Staubli VAL3: tool.pjx

--- tool.pjx ---
Parameters version=s7.2.1 stackSize=5000 millimeterUnit=true
Program file=buildList.pgx
Program file=editAction.pgx
Program file=editTool.pgx
Program file=insertInstr.pgx
Program file=listAdd.pgx
Program file=loadPage.pgx
Program file=main.pgx
Program file=onBackSpace.pgx
Program file=onEnterEvent.pgx
Program file=onExit.pgx
Program file=onF1Event.pgx
Program file=onF2Event.pgx
Program file=onF3Event.pgx
Program file=onF4Event.pgx
Program file=onF5Event.pgx
Program file=onF6Event.pgx
Program file=onF7Event.pgx
Program file=onF8Event.pgx
Program file=onStart.pgx
Program file=refresh.pgx
Program file=refreshAction.pgx
Program file=refreshDynamic.pgx
Program file=refreshStatic.pgx
Data file=tool.dtx
Library alias=io path=Disk://io/io.pjx
Library alias=page path=Disk://kernel/template/page/page.pjx
Library alias=use path=Disk://kernel/userPage/userPage.pjx
Library alias=language path=Disk://kernel/language/language.pjx
Library alias=tcp path=Disk://kernel/tool/tool.pjx

--- tool.dtx ---
num nIndex
num nIndexTool
num nKey
public num nPage
num nRefresh
num nTime = 1
num nView
string sEvent
public string sItems
string sList
string sMenu
string sMessage
string sMenu8[8]
string sActionON[3]
string sActionOFF[3]
bool bButton[8]
bool bLarge

--- main.pgx ---
public program main()
  local tool l_tTool
  local num l_nSize
  local bool l_bSave
  local num l_nStatus
  local bool l_bToReset
  local bool l_bCalcolate
  local frame l_fNewWorld
begin
  // INIT
  call onStart()
  // LOOP UNTIL nKey=255
  do
    call tcp:getSize(l_nSize)
    call tcp:getTool(l_tTool,nIndexTool)
    call refresh()
    if l_bCalcolate
      $jogContext(l_tTool,world,0)
      l_bCalcolate=false
    endIf
    nKey=getKey()
    // tool setting

    // list....
    call use:listevent(nKey,nIndex,sEvent)
    nView=use:nView
    switch nKey
      case 263
        // BACKSPACE
        call onBackSpace(l_tTool)
        l_bCalcolate=true
        l_bSave=true
      break
      case 264
        // LEFT CLICK -1
        if nIndexTool>0
          nIndexTool=nIndexTool-1
          l_bSave=true
          l_bCalcolate=true
        endIf
      break
      case 268
        // RIGHT CLICK +1
        if nIndexTool<l_nSize-1
          nIndexTool=nIndexTool+1
          l_bSave=true
          l_bCalcolate=true
        endIf
      break
      case 271
        call onF1Event()
      break
      case 272
        call onF2Event()
      break
      case 273
        // HERE
        call onF3Event(l_bSave)
      break
      case 274
        // COMPUTE
        call onF4Event(l_bSave)
        l_bCalcolate=true
      break
      case 275
        // MOVE
        call onF5Event()
      break
      case 276
        // DUPLICATE
        call onF6Event(l_tTool.trsf,l_bSave)
      break
      case 277
        // DELETE
        call onF7Event(l_bSave)
      break
      case 278
        // NEW
        call onF8Event(l_bSave)
      break
      case 270
        // USE ALSO BACKSPACE
        // EDIT FIELD
        call onEnterEvent(l_tTool)
        l_bCalcolate=true
        l_bSave=true
      break
    endSwitch
    // release the resource
    delay(0)
  until nKey==255
  // on Exit
  $jogContext(l_tTool,world,0)
  call onExit(l_bSave)
end

--- buildList.pgx ---
program buildList()
  local num l_nSize
  local string l_sName
  local num i
  local string l_sMessage
  local tool l_tTool
  local string l_sString
begin
  // INIT the list
  l_sString=""
  call use:stringCopy(l_sString,sList)
  //
  // Build the list
  //
  // get the GUN
  call tcp:getTool(l_tTool,nIndexTool)
  // show the gun
  call tcp:getName(l_sName,nIndexTool)
  call language:message(l_sMessage,21)
  l_sName=l_sMessage+"> "+l_sName
  // create the list
  call listAdd(l_sName)
  call listAdd("coord  X > "+toString(".2",l_tTool.trsf.x))
  call listAdd("coord  Y > "+toString(".2",l_tTool.trsf.y))
  call listAdd("coord  Z > "+toString(".2",l_tTool.trsf.z))
  call listAdd("coord RX > "+toString(".2",l_tTool.trsf.rx))
  call listAdd("coord RY > "+toString(".2",l_tTool.trsf.ry))
  call listAdd("coord RZ > "+toString(".2",l_tTool.trsf.rz))
  // TCP ON OFF
  call language:message(l_sMessage,123)
  call use:strfill(l_sMessage,9,l_sMessage)
  call listAdd(l_sMessage+"> ON ")
  call listAdd(l_sMessage+"> OFF")
end

--- editAction.pgx ---
program editAction(string& x_sAction[], bool& x_bSave[])
  local string l_sMessage
  local string l_sAction[3]
  local string l_sInstruction
  local bool l_bYes
  local num i
  local num l_nKey
  local num l_nIndex
  local string l_sButton[2]
  local string l_sString
begin
  // make a copy
  call use:stringCopy(x_sAction,l_sAction)
  // refresh
  call refreshAction(l_nIndex,x_sAction)
  // loop
  do
    l_nKey=getKey()
    l_sString=""
    call use:listevent(l_nKey,l_nIndex,l_sString)
    if l_nKey==270
      //
      //  edit the instruction
      //
      // insert a new one
      if l_sAction[l_nIndex]==""
        call insertInstr(l_sMessage)
        if l_sMessage!=""
          l_sAction[l_nIndex]=l_sMessage
        endIf
      else
        // delete
        call language:message(l_sMessage,171)
        // get the yes_no button
        call language:getYesNo(l_sButton)
        // ask the question
        call use:yes_no(l_sMessage,l_sButton,l_bYes)
        if l_bYes
          l_sAction[l_nIndex]=""
        endIf
      endIf
      // copy back
      l_sInstruction=""
      if l_sAction[0]!="" or l_sAction[1]!="" or l_sAction[2]!=""
        for i=0 to 1
          l_sInstruction=l_sInstruction+l_sAction[i]+"^"
        endFor
        l_sInstruction=l_sInstruction+l_sAction[2]
      endIf
      // refresh
      call refreshAction(l_nIndex,l_sAction)
    endIf
    delay(0)
    // use left to go bak or escape to no validate
  until l_nKey==264 or l_nKey==255 or l_nKey==278
  //
  if l_nKey!=255
    x_bSave=true
    call use:stringCopy(l_sAction,x_sAction)
  endIf
end

--- editTool.pgx ---
program editTool(trsf& x_tTrsf[])
  local num i
  local num l_nX
  local num l_nY
  local bool l_bEdit
  local string l_sString
begin
  //
  //  search the ">" to change the right side from here of the the string
  //
  call use:getListPosition(l_nX,l_nY)
  //i=find(sEvent,">")
  call use:findPos(sEvent,">",i)
  // clean the line
  call use:listcursor(use:nView,false)
  // read the name
  if i!=-1 and nIndex==0
    sEvent=right(sEvent,getDisplayLen(sEvent)-i-2)
    // read the name
    call use:read(i+l_nX+1,1,sEvent,10,false)
  endIf
  l_sString=""
  switch nIndex
    case 0
      if nIndexTool!=-1
        call tcp:setName(sEvent,nIndexTool)
      endIf
    break
    case 1
      //
      //  x-value
      //

      call use:changeValue(x_tTrsf.x,0,0,i+40-use:nBottomX+1,use:nView+1,l_sString)
    break
    case 2
      //
      //  y-value
      //
      call use:changeValue(x_tTrsf.y,0,0,i+40-use:nBottomX+1,use:nView+1,l_sString)
    break
    case 3
      //
      //  z-value
      //
      call use:changeValue(x_tTrsf.z,0,0,i+40-use:nBottomX+1,use:nView+1,l_sString)
    break
    case 4
      //
      //  rx-value
      //
      call use:changeValue(x_tTrsf.rx,0,0,i+40-use:nBottomX+1,use:nView+1,l_sString)
    break
    case 5
      //
      //  ry-value
      //
      call use:changeValue(x_tTrsf.ry,0,0,i+40-use:nBottomX+1,use:nView+1,l_sString)
    break
    case 6
      //
      //  rz-value
      //
      call use:changeValue(x_tTrsf.rz,0,0,i+40-use:nBottomX+1,use:nView+1,l_sString)
    break
    case 7
      //
      // change the ACTION ON
      //
      call editAction(sActionON,l_bEdit)
      if l_bEdit
        call tcp:setAction(sActionON,nIndexTool,true)
      endIf
    break
    case 8
      //
      // change the ACTION OFF
      //
      call editAction(sActionOFF,l_bEdit)
      if l_bEdit
        call tcp:setAction(sActionOFF,nIndexTool,false)
      endIf
    break
  endSwitch
end

--- insertInstr.pgx ---
program insertInstr(string& x_sItem[])
  local num i
  local num l_nNum
begin
  // TODO
  call use:setSizeList(14,0,10,11)
  call use:setView(false)
  call use:listcreate("Select")
  // insert the action on Point

  call use:listupdate(0)
  // SELECT THE ITEM
  x_sItem=""
  do
    i=getKey()
    l_nNum=0
    call use:listevent(i,l_nNum,x_sItem)
    delay(0)
  until i==255 or i==270
  //

  // NOT GOOD
  x_sItem=""
end

--- listAdd.pgx ---
program listAdd(string x_sEvent)
begin
  // add in the queue
  if sList!=""
    $dins(sList,size(sList))
  endIf
  sList[size(sList)-1]=x_sEvent
end

--- loadPage.pgx ---
program loadPage(string x_sPage, string& x_sItems[])
// load the next page
  local num i
  local string l_sMessage
begin
  // look if the page libload is correct
  i=page:libLoad(x_sPage)
  if i!=0
    logMsg("[VALlaser] INTERFACE:PAGE LIBLOAD "+x_sPage+" result "+toString("",i))
    call language:message(l_sMessage,-7)
    popUpMsg(l_sMessage+x_sPage+" ; "+toString("",i))
  else
    // copy all the field from x_sItems to the next page
    call use:stringCopy(x_sItems,page:sItems)
    call page:main()
    // to give back
    call use:stringCopy(page:sItems,x_sItems)
  endIf
end

--- onBackSpace.pgx ---
program onBackSpace(tool& x_tTool[])
begin
  //
  // NB sEvent is the selected
  // element in the LIST
  //
  if nIndex==0
    call editTool(x_tTool.trsf)
    call tcp:setTool(x_tTool,nIndexTool)
    logMsg("[VALlaser] INTERFACE:Change value of the tool :"+toString("",nIndexTool))
  endIf
  //
end

--- onEnterEvent.pgx ---
program onEnterEvent(tool& x_tTool[])
begin
  //
  // NB sEvent is the selected
  // element in the LIST
  //
  call editTool(x_tTool.trsf)
  call tcp:setTool(x_tTool,nIndexTool)
  logMsg("[VALlaser] INTERFACE:Change value of the tool :"+toString("",nIndexTool))
  //
end

--- onExit.pgx ---
program onExit(bool x_bSave)
  local string l_sMessage
  local bool l_bYes
  local num l_nResult
begin
  if x_bSave
    // ask to save
    //    call language:message(l_sMessage,-1)
    //    call use:yes_no(l_sMessage,l_bYes)
    //    if l_bYes
    call tcp:save(l_nResult)
    // send back the gun
    //    endIf
  endIf
  // give back and update

end

--- onF1Event.pgx ---
program onF1Event()
begin
  // look if the bButton is enable
  if bButton[0]
    //
  endIf
end

--- onF2Event.pgx ---
program onF2Event()
begin
  // look if the bButton is enable
  if bButton[1]
    //
  endIf
end

--- onF3Event.pgx ---
program onF3Event(bool x_bSave)
  local string l_sMessage
  local bool l_bYes
  local string l_sButton[2]
begin
  // look if the bButton is enable
  if bButton[2]
    //
    if nIndexTool==0
      call language:message(l_sMessage,125)
      // get the yes_no button
      call language:getYesNo(l_sButton)
      // ask the question
      call use:yes_no(l_sMessage,l_sButton,l_bYes)
      if l_bYes
        call tcp:here()
        call language:message(l_sMessage,121)
        popUpMsg(l_sMessage)
        logMsg("[VALlaser] INTERFACE:Take the reference point")
        x_bSave=true
      endIf
    endIf
  endIf
end

--- onF4Event.pgx ---
program onF4Event(bool& x_bSave[])
  local bool l_bCheck
  local tool l_tTool
  local string l_sMessage
  local frame l_fNewWorld
begin
  // look if the bButton is enable
  if bButton[3]
    //

      if nIndexTool!=0
        call tcp:checkPoint(l_bCheck)
        if l_bCheck
          call tcp:compose(nIndexTool)
          call tcp:getTool(l_tTool,nIndexTool)
          $jogContext(l_tTool,world,0)
          logMsg("[VALlaser] INTERFACE:Compose the gun")
          x_bSave=true
        else
          call language:message(l_sMessage,122)
          popUpMsg(l_sMessage)
        endIf
      endIf

  endIf
end

--- onF5Event.pgx ---
program onF5Event()
  local bool l_bCheck
  local string l_sMessage
begin
  // look if the bButton is enable
  if bButton[4]
    //
    if workingMode()==1
      resetMotion()
      call tcp:checkPoint(l_bCheck)
      if l_bCheck
        call language:message(l_sMessage,203)
        call tcp:goToPoint(nIndexTool)
        logMsg("[VALlaser] INTERFACE:Go to the reference Point")
        call use:timerDialog(l_sMessage,2)
      endIf
    endIf
  endIf
end

--- onF6Event.pgx ---
program onF6Event(trsf x_tTrsf, bool& x_bSave[])
  local string l_sMessage
  local string l_sName
  local num l_nSize
begin
  // look if the bButton is enable
  if bButton[5]
    //
    // DUPLICATE
    //
    call language:message(l_sMessage,126)
    call tcp:getName(l_sName,nIndexTool)
    popUpMsg(l_sMessage+l_sName)
    call tcp:new(x_tTrsf)
    call tcp:getSize(l_nSize)
    nIndexTool=l_nSize-1
    // refresh and modify the name
    call buildList()
    call refreshStatic()
    nIndex=0
    call editTool(x_tTrsf)
    logMsg("[VALlaser] INTERFACE:Insert new tool at index: "+toString("",l_nSize))
    x_bSave=true
  endIf
end

--- onF7Event.pgx ---
program onF7Event(bool& x_bSave[])
  local string l_sMessage
  local bool l_bFound
  local string l_sTrajName
  local bool l_bYes
  local string l_sString
  local string l_sButton[2]
begin
  // look if the bButton is enable
  if bButton[6]
    // delete the selected tool
    if  nIndexTool!=0
      call language:message(l_sMessage,120)
      // get the yes_no button
      call language:getYesNo(l_sButton)
      // ask the question
      call use:yes_no(l_sMessage+toString("",nIndexTool),l_sButton,l_bYes)
      if l_bYes
        call refreshStatic()

        if !l_bFound
          // move from the all traj the indexTool

          call tcp:delete(nIndexTool)
          nIndexTool=nIndexTool-1
          logMsg("[VALlaser] INTERFACE:Delete the tool: "+toString("",nIndexTool))
          x_bSave=true
        else
          // show the message the tool is already used
          call language:message(l_sMessage,124)
          call language:message(l_sString,29)
          popUpMsg(l_sMessage+l_sString+l_sTrajName)
        endIf
      endIf
    endIf
  endIf
end

--- onF8Event.pgx ---
program onF8Event(bool& x_bSave[])
  local trsf l_tEmpty
  local num l_nSize
begin
  // look if the bButton is enable
  if bButton[7]
    //
    l_tEmpty={0,0,0,0,0,0}
    call tcp:new(l_tEmpty)
    call tcp:getSize(l_nSize)
    nIndexTool=l_nSize-1
    // refresh and modify the name
    call buildList()
    call refreshStatic()
    nIndex=0
    sEvent=""
    call editTool(l_tEmpty)
    logMsg("[VALlaser] INTERFACE:Insert new tool at index: "+toString("",l_nSize))
    x_bSave=true
  endIf
end

--- onStart.pgx ---
program onStart()
  local num i
  local string l_sMessage
begin
  // logMsg
  logMsg("[VALlaser] INTERFACE:PAGE TOOL")
  // be aware these value will change all the value
  call language:message(l_sMessage,129)
  popUpMsg(l_sMessage)
  // set the tool as default

  // restore the old value

  // reset the Key pressure
  call use:nullKey(nKey)
  // define the list
  call buildList()
  // build the page
  call refreshStatic()
  // define the list
end

--- refresh.pgx ---
program refresh()
// // page refresh
begin
  // refresh the static message
  if (nKey>=270 and nKey<=278) or nKey==268 or nKey==264 or use:bUseRefresh
    call buildList()
    call refreshStatic()
    call refreshDynamic()
  else
    // refresh the Dynamic message
    if (clock()-nRefresh>nTime)
      call refreshDynamic()
    endIf
  endIf
  // release the resource
  delay(0)
end

--- refreshAction.pgx ---
program refreshAction(num x_nIndex, string& x_sAction[])
  local string l_sMessage
  local string l_sTitle
  local string l_sComment
  local num i
  local string l_sAction[3]
  local num l_nSize
begin
  //
  // INSTRUCTION
  //
  cls()
  // create a menu to edit the action
  call use:setSizeList(5,3,30,3)
  call use:setView(false)
  // show the title
  call tcp:getSize(l_nSize)
  call language:message(l_sMessage,124)
  l_sTitle=l_sMessage+toString("3",nIndexTool)+"/"+toString("",l_nSize-1)
  call tcp:getName(l_sMessage,nIndexTool)
  l_sTitle=l_sTitle+" "+l_sMessage
  call use:listcreate(l_sTitle)
  // get the action string
  call language:message(l_sMessage,176)
  // insert all the 3 action
  for i=0 to 2
    call use:listadd(l_sMessage+toString("",i+1)+"> "+x_sAction[i])
  endFor
  // show it
  call use:clear(0,13)
  call use:typeMenu(8,"OK")
  use:nView=x_nIndex
  call use:listupdate(0)
  //
end

--- refreshDynamic.pgx ---
program refreshDynamic()
begin
  // DO NOT CHANGE
  nRefresh=clock()
  use:bUseRefresh=false
  //
  // ADD HERE
  //
end

--- refreshStatic.pgx ---
program refreshStatic()
  local num l_nSize
  local string l_sMessage
  local string l_sTitle
  local string l_sInstruction
  local num i
begin
  cls()
  //
  // set the view of the use:nPage..
  //
  // SET THE use:nPage NUMBER
  use:nPage=1400
  //
  if nIndexTool==0
    use:nPage=use:nPage+6
  endIf

  // USE <>PROFILE for <>nPage

  // load the menu page

    call language:page(l_sMessage,use:nPage)
    // define the menu
    call use:stringToArray(l_sMessage,sMenu)
    call use:setMenu(sMenu,true,2)

  //
  call use:getMenu(sMenu,bButton)
  //
  // CREATE THE LIST
  //
  // define your list size for default
  call use:setSizeList(19,0,19,9)
  call use:setView(bLarge)
  //
  call tcp:getSize(l_nSize)
  call language:message(l_sTitle,124)
  l_sTitle=l_sTitle+toString("3",nIndexTool)+"/"+toString("",l_nSize-1)
  call use:listcreate(l_sTitle)
  // insert inside the list
  call use:listadd(sList)
  // show the instruction ON
  call tcp:getAction(sActionON,true,nIndexTool)
  l_sInstruction=sActionON
  for i=1 to size(sActionON)-1
    if sActionON[i]!=""
      l_sInstruction=l_sInstruction+"·"+sActionON[i]
    endIf
  endFor
  call use:typeLen(0,11,"ON >"+l_sInstruction,40)
  // show the instruction OFF
  call tcp:getAction(sActionOFF,false,nIndexTool)
  // array to string
  l_sInstruction=sActionOFF
  for i=1 to size(sActionOFF)-1
    if sActionOFF[i]!=""
      l_sInstruction=l_sInstruction+"·"+sActionOFF[i]
    endIf
  endFor
  call use:typeLen(0,12,"OFF>"+l_sInstruction,40)
  //
  // refresh the cursor
  use:nView=nView
  // refresh the list
  call use:listupdate(nIndex-nView)
end
